FUNCTION_BLOCK Train1
  (* Standard: 61499-2 *)
  (* Version 0,1, 2015-00-24, Th?o, PC_THEO *)
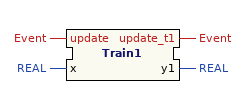
  EVENT_INPUT
    update;
  END_EVENT
  EVENT_OUTPUT
    update_t1;
  END_EVENT
  VAR_INPUT
    x : REAL;
  END_VAR
  VAR_OUTPUT
    y1 : REAL;
  END_VAR
  VAR
    d : REAL;
    k : INT;
    C1y1 : REAL;
    delta : REAL;
  END_VAR
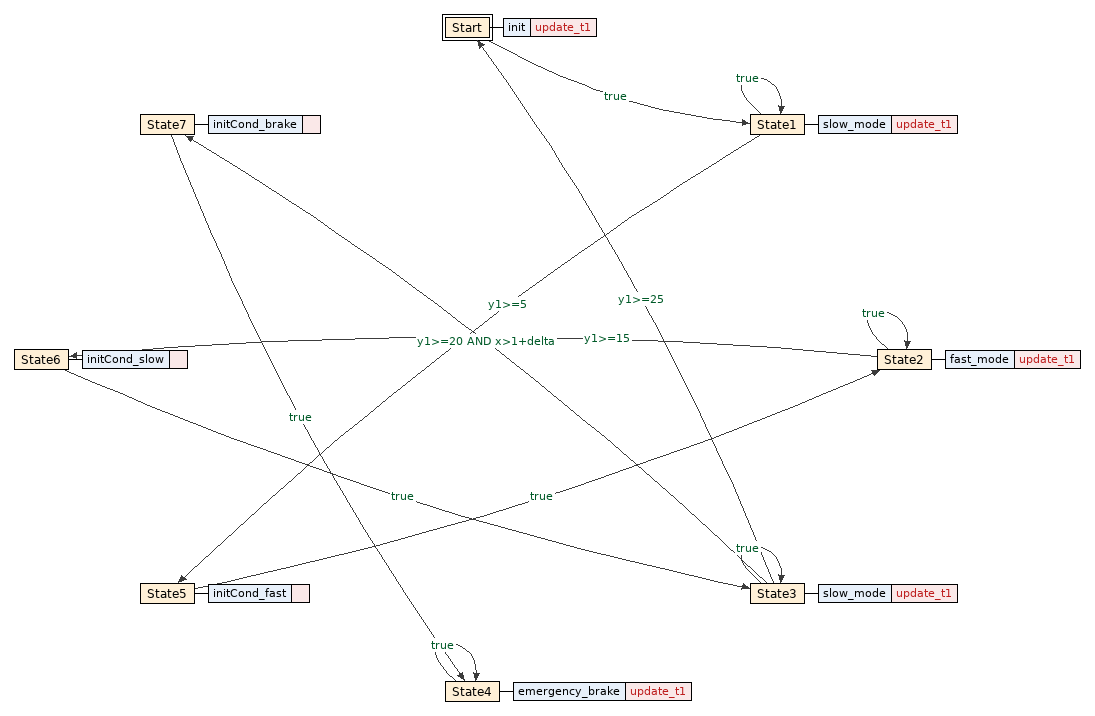
  EC_STATES
    Start : init -> update_t1;
    State1 : slow_mode -> update_t1;
    State2 : fast_mode -> update_t1;
    State3 : slow_mode -> update_t1;
    State4 : emergency_brake -> update_t1;
    State5 : initCond_fast;
    State6 : initCond_slow;
    State7 : initCond_brake;
  END_STATES
  EC_TRANSITIONS
    Start TO State1 := true;
    State1 TO State5 := y1>=5;
    State1 TO State1 := true;
    State2 TO State6 := y1>=15;
    State2 TO State2 := true;
    State3 TO State7 := y1>=20 AND x>1+delta;
    State3 TO Start := y1>=25;
    State3 TO State3 := true;
    State4 TO State4 := true;
    State5 TO State2 := true;
    State6 TO State3 := true;
    State7 TO State4 := true;
  END_TRANSITIONS
  ALGORITHM init IN C:
me->y1=0;
me->delta=0.0001;
me->k=1;
me->C1y1=-1;
  END_ALGORITHM
  ALGORITHM slow_mode IN C:
me->y1=me->C1y1*exp(-1.0L/2.0L*me->d*me->k)+1;
(me->k)++;
  END_ALGORITHM
  ALGORITHM fast_mode IN C:
me->y1=me->C1y1*exp(-1*me->d*me->k)+2;
(me->k)++;
  END_ALGORITHM
  ALGORITHM emergency_brake IN C:
me->y1=me->C1y1*exp(-1.0L/10.0L*me->d*me->k);
(me->k)++;

if (me->y1 <= me->delta) {
	printf ("Emergency brake : Train stopped at y1 = %f and x = %f\n",me->y1, me->x);
	exit(1);
	}
  END_ALGORITHM
  ALGORITHM initCond_fast IN C:
me->k=1;
me->C1y1=me->x-2;
printf("fast mode on\n");
  END_ALGORITHM
  ALGORITHM initCond_slow IN C:
me->k=1;
me->C1y1=me->x-1;
printf("slow mode on\n");
  END_ALGORITHM
  ALGORITHM initCond_brake IN C:
me->k=1;
me->C1y1=me->x-10;
printf("Emergency brake !!!\n");
  END_ALGORITHM
END_FUNCTION_BLOCK
